# EPICS autosave request: iocBoot/iocLinux/DSA2000_settings.req
file "mca_settings.req",          P=$(P), M=aim_adc1
file "icbDsp_settings.req",       P=$(P), DSP=dsp1
file "DSA2000_HVPS_settings.req", P=$(P), HVPS=hvps1:
